// Mitsubishi GX Works2 project: GT_EX2+   PLC: Q03UDV

PROGRAM MAIN
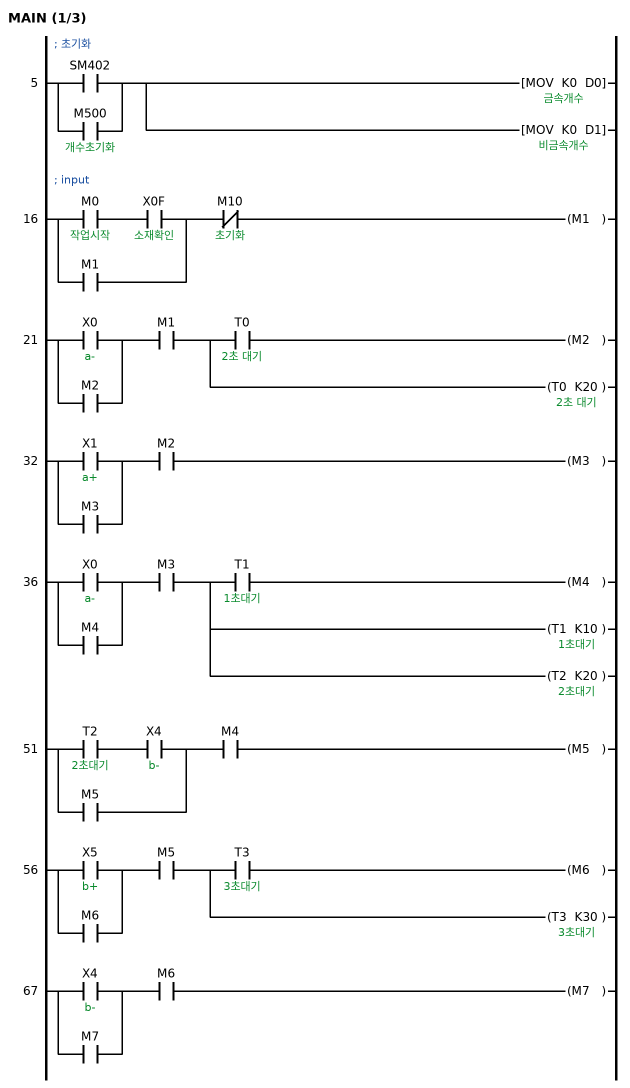
; 초기화
5     LD      SM402
      OR      M500  ; 개수초기화
      MOV     K0 D0  ; 금속개수
      MOV     K0 D1  ; 비금속개수
; input
16    LD      M0  ; 작업시작
      AND     X0F  ; 소재확인
      OR      M1
      ANI     M10  ; 초기화
      OUT     M1
21    LD      X0  ; a-
      OR      M2
      AND     M1
      MPS
      AND     T0  ; 2초 대기
      OUT     M2
      MPP
      OUT     T0 K20  ; 2초 대기
32    LD      X1  ; a+
      OR      M3
      AND     M2
      OUT     M3
36    LD      X0  ; a-
      OR      M4
      AND     M3
      MPS
      AND     T1  ; 1초대기
      OUT     M4
      MPP
      OUT     T1 K10  ; 1초대기
      OUT     T2 K20  ; 2초대기
51    LD      T2  ; 2초대기
      AND     X4  ; b-
      OR      M5
      AND     M4
      OUT     M5
56    LD      X5  ; b+
      OR      M6
      AND     M5
      MPS
      AND     T3  ; 3초대기
      OUT     M6
      MPP
      OUT     T3 K30  ; 3초대기
67    LD      X4  ; b-
      OR      M7
      AND     M6
      OUT     M7
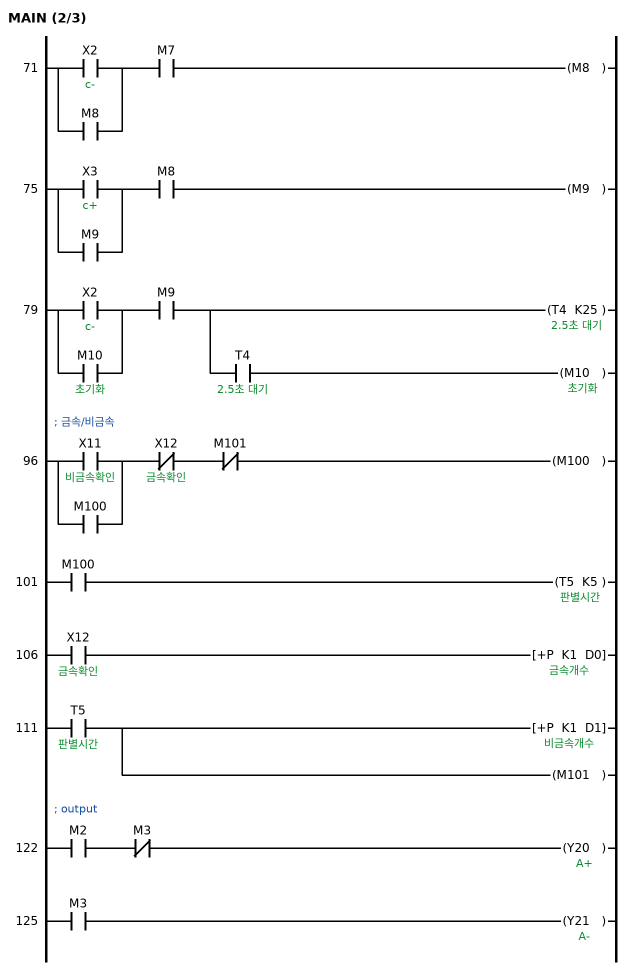
71    LD      X2  ; c-
      OR      M8
      AND     M7
      OUT     M8
75    LD      X3  ; c+
      OR      M9
      AND     M8
      OUT     M9
79    LD      X2  ; c-
      OR      M10  ; 초기화
      AND     M9
      OUT     T4 K25  ; 2.5초 대기
      AND     T4  ; 2.5초 대기
      OUT     M10  ; 초기화
; 금속/비금속
96    LD      X11  ; 비금속확인
      OR      M100
      ANI     X12  ; 금속확인
      ANI     M101
      OUT     M100
101   LD      M100
      OUT     T5 K5  ; 판별시간
106   LD      X12  ; 금속확인
      +P      K1 D0
111   LD      T5  ; 판별시간
      +P      K1 D1
      OUT     M101
; output
122   LD      M2
      ANI     M3
      OUT     Y20  ; A+
125   LD      M3
      OUT     Y21  ; A-
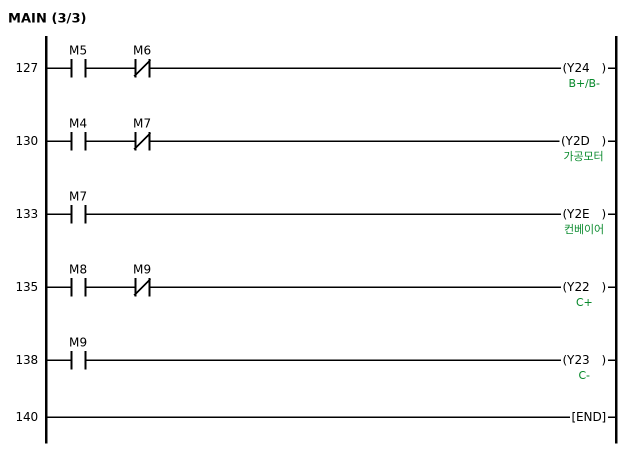
127   LD      M5
      ANI     M6
      OUT     Y24  ; B+/B-
130   LD      M4
      ANI     M7
      OUT     Y2D  ; 가공모터
133   LD      M7
      OUT     Y2E  ; 컨베이어
135   LD      M8
      ANI     M9
      OUT     Y22  ; C+
138   LD      M9
      OUT     Y23  ; C-
140   END
END_PROGRAM
